(* PLC project  *)

PROGRAM MainRoutine

(* LD diagram, written out as Structured Text *)
END_PROGRAM
